FUNCTION_BLOCK List
VAR_GENERIC CONSTANT
	ListSize : UDINT := 2;
END_VAR
EXTENDS Collection<ListSize> IMPLEMENTS I_List
VAR
	_ListCount : UDINT := 0;
END_VAR

METHOD AddItem
VAR_INPUT
	Item : I_Base;
END_VAR
SUPER^.AddItem(Item);
CountListItems();
END_METHOD

METHOD Clear
SUPER^.Clear();
CountListItems();
END_METHOD

METHOD ContainsItem : BOOL
VAR_INPUT
	Item : I_Base;
END_VAR

VAR
	i	  : UDINT;
	pItem : POINTER TO I_Base;
END_VAR
IF Item = 0 THEN
	Trace.LogMessage(InstancePath, 'Item is not a valid interface!');
	RETURN;
END_IF

IF _ListCount = 0 THEN
	RETURN;
END_IF

FOR i := 0 TO (_ListCount - 1) DO
	IF _Data[i] = Item AND _Data[i] <> 0 THEN
		ContainsItem := TRUE;
		RETURN;
	END_IF
END_FOR
END_METHOD

{attribute 'monitoring' := 'call'}
PROPERTY Count : UDINT
GET
Count := _ListCount;
END_GET
END_PROPERTY

METHOD PRIVATE CountListItems
VAR
	i	  : UDINT;
	pItem : POINTER TO I_Base;
END_VAR
IF _Count = 0 THEN
	_ListCount := 0;
	RETURN;
END_IF

_ListCount := 0;
FOR i := 0 TO (_Count - 1) DO
	IF _Data[i] <> 0 THEN
		_ListCount := _ListCount + 1;
	END_IF
END_FOR
END_METHOD

METHOD GetAtIndex : I_Base
VAR_INPUT
	Index : UDINT;
END_VAR

VAR
	pItem : POINTER TO I_Base;
END_VAR
IF Count = 0 THEN
	Trace.LogMessage(InstancePath, 'No Items found in this List!');
	RETURN;
END_IF

IF Index > (_Count - 1) THEN
	Trace.LogMessage(InstancePath, 'Index does not exist in List!');
	RETURN;
END_IF

GetAtIndex := _Data[Index];
END_METHOD

METHOD InsertAtIndex : BOOL
VAR_INPUT
	Item  : I_Base;
	Index : UDINT;
END_VAR

VAR
	pItem	  : POINTER TO I_Base;
	pItemNext : POINTER TO I_Base;
	i		  : UDINT;
END_VAR
IF Index > _Count THEN
	InsertAtIndex := FALSE;
	RETURN;
END_IF

_Count := (_Count + 1);
FOR i := _Count TO Index + 1 BY -1 DO
	_Data[i] := _Data[i - 1];
END_FOR

_Data[Index] := Item;
CountListItems();
END_METHOD

METHOD RemoveAtIndex
VAR_INPUT
	Index : UDINT;
END_VAR

VAR
	pItem : POINTER TO I_Base;
END_VAR
IF Count = 0 THEN
	Trace.LogMessage(InstancePath, 'No Items found in this List!');
	RETURN;
END_IF

IF Index > (_Count - 1) THEN
	Trace.LogMessage(InstancePath, 'Index does not exist in List!');
	RETURN;
END_IF

MEMMOVE(ADR(_Data[Index]), ADR(_Data[Index + 1]), (_Count - Index - 1) * SIZEOF(PVOID));
_Count := _Count - 1;

//pItem  := Collection.pBuffer + (Index * SIZEOF(PVOID));
CountListItems();
END_METHOD

METHOD RemoveItem
VAR_INPUT
	Item : I_Base;
END_VAR

VAR
	pItem		 : POINTER TO I_Base;
	pItemNext	 : POINTER TO I_Base;
	i			 : UDINT;
	removedItems : UDINT;
END_VAR
IF _Count = 0 THEN
	Trace.LogMessage(InstancePath, 'No Items found in this Collection!');
	RETURN;
END_IF

IF Item = 0 THEN
	Trace.LogMessage(InstancePath, 'Item to remove needs to be valid interface!');
	RETURN;
END_IF

FOR i := 0 TO (_Count - 1) DO
	IF _Data[i] = Item THEN
		_Data[i]	 := 0;
		removedItems := removedItems + 1;
	END_IF
END_FOR

IF _Count > 1 THEN
	FOR i := 0 TO (_Count - 2) DO
		IF _Data[i] = 0 AND _Data[i + 1] <> 0 THEN
			_Data[i]	 := _Data[i + 1];
			_Data[i + 1] := 0;
		END_IF
	END_FOR
END_IF

CountListItems();
_Count := _Count - removedItems;
END_METHOD

END_FUNCTION_BLOCK

(* stored: Version 1.1.0.1, ProductVersion 3.1.4026.18
   POU List: Id {af29319b-574f-4e46-9fab-e40ca5d32152}, SpecialFunc None
   Folder Collection: Id {2b9c8ba3-c154-494a-a636-238324b2aea7}
   Folder Private: Id {a679ba01-c874-4153-a7ec-1396e367be78}
   Method AddItem: Id {1596be71-9d81-43cb-8891-f42b67f8ce52}
   Method Clear: Id {44514f62-79d4-4e53-bbe0-4cc03497e90d}
   Method ContainsItem: Id {4cfb3b5d-edfb-4547-a262-8c17ef4c6601}
   Property Count: Id {f6eb0ff9-dee3-4c0e-a279-9a01659a8597}
   Get Get: Id {0fba2825-bfa9-4b65-a5b6-25c736c60f27}
   Method CountListItems: Id {9a734140-c852-430b-8cdb-5e1e55a05c3d}
   Method GetAtIndex: Id {6175e397-7fb9-4a5f-b2c9-81e015814843}
   Method InsertAtIndex: Id {3d241dbc-f3ba-4d49-852a-1cfd8db3a81f}
   Method RemoveAtIndex: Id {12021925-b0b2-4465-b4f0-31cc3667b43a}
   Method RemoveItem: Id {cd74e3fb-92ab-435b-829f-468f2665dfb1} *)
